FUNCTION_BLOCK INTERNAL FINAL FB_WriteRepeatedFieldInt32Tests EXTENDS FB_TestSuite
VAR_INPUT
END_VAR
VAR_OUTPUT
END_VAR
VAR
	fbFieldCodec : FB_FieldCodecInt32(nTag:= 0);
	aActual    	 : ARRAY [0..7] OF DINT;
	fbRepeatedField		: FB_RepeatedField(anyArray:= F_ToAnyType(aActual), anyFirstElem:= F_ToAnyType(aActual[0]), ipFieldCodec:= fbFieldCodec);
END_VAR

ShouldWriteRepeatedFieldTheory();

METHOD PRIVATE Reset
VAR_INPUT
END_VAR
fbRepeatedField.Initialize();
MEMSET(destAddr:= ADR(aActual), fillByte:= 16#0, n:= SIZEOF(aActual));
END_METHOD

METHOD PRIVATE ShouldWriteRepeatedField
VAR_IN_OUT CONSTANT
    aExpected   : ARRAY [*] OF BYTE;
END_VAR
VAR_INPUT
    aValues     : ARRAY [0..7] OF DINT;
    nLength     : UDINT;
    nTag        : UDINT;
    nBufferPosStart     : UDINT;
    nExpectedBufferPos  : UDINT;
    ipFieldCodec        : I_FieldCodec;
END_VAR
VAR_INST
    fbCtx   : FB_WriteContext;
END_VAR
VAR
    aActualBuffer       : ARRAY [0..63] OF BYTE;
    hr                  : HRESULT;

END_VAR
// Arrange
Reset();
fbCtx.FromBuffer(aActualBuffer);
fbCtx.refCtx.stState.nBufferPos := nBufferPosStart;
ipFieldCodec.Tag := nTag;
fbRepeatedField.InitializeFromArray(anyArray:= F_ToAnyType(aValues), anyFirstElem:= F_ToAnyType(aValues[0]), nCount:= nLength);

// Act
hr := fbRepeatedField.WriteTo(fbWriteCtx:= fbCtx, ipFieldCodec:= ipFieldCodec);

// Assert
AssertEquals_DINT(
    Expected:= S_OK,
    Actual:= hr,
    Message:= 'Expected S_OK instead of error');
    
{warning disable C0041}
AssertArrayEquals_BYTE(Expecteds:= aExpected, Actuals:= aActualBuffer, Message:= '');
 
AssertEquals_UDINT(
    Expected:= nExpectedBufferPos,
    Actual:= fbCtx.refCtx.stState.nBufferPos,
    Message:= CONCAT('Expected stState.nBufferPos to equal ', TO_STRING(nExpectedBufferPos)));
END_METHOD

METHOD PRIVATE ShouldWriteRepeatedFieldTheory : REFERENCE TO FB_Test
VAR CONSTANT
    cRawValueZeroLength     : ARRAY[0..63] OF BYTE := [16#00, 16#00];
    cRawValue1              : ARRAY[0..63] OF BYTE := [16#00, 16#0A, 16#18, 16#00, 16#D2, 16#09, 16#B9, 16#0A, 16#FF, 16#FF, 16#FF, 16#FF, 16#FF, 16#FF, 16#FF, 16#FF, 16#FF, 16#01, 16#CE, 16#C2, 16#F1, 16#05, 16#FF, 16#FF, 16#FF, 16#FF, 16#07];  
END_VAR

VAR CONSTANT
    aExpectedZeroLength     : ARRAY [0..7] OF DINT := [0, 0, 0, 0, 0, 0, 0, 0];
    aExpected1              : ARRAY [0..7] OF DINT := [0, 1234, 1337, -1, 12345678, 2147483647];
END_VAR
TEST(__POUNAME());

ShouldWriteRepeatedField(aExpected:= cRawValueZeroLength, aValues:= aExpectedZeroLength, nLength:= 0, nTag:= F_MakeTag(1, E_WireType.LengthDelimited), nBufferPosStart:= 0, nExpectedBufferPos:= 0, ipFieldCodec:= THIS^.fbFieldCodec);
ShouldWriteRepeatedField(aExpected:= cRawValue1, aValues:= aExpected1, nLength:= 6, nTag:= F_MakeTag(1, E_WireType.LengthDelimited), nBufferPosStart:= 1, nExpectedBufferPos:= 27, ipFieldCodec:= THIS^.fbFieldCodec);

TEST_FINISHED_NAMED(__POUNAME());
END_METHOD

END_FUNCTION_BLOCK

(* stored: Version 1.1.0.1
   POU FB_WriteRepeatedFieldInt32Tests: Id {bc593a6b-e6cc-4be6-a6ba-0b0aa8d4d524}, SpecialFunc None
   Method Reset: Id {1c3d5621-576c-4b6d-9236-b5891ede49f2}
   Method ShouldWriteRepeatedField: Id {320e051d-b81f-4409-b73c-7f1b4d7dc30b}
   Method ShouldWriteRepeatedFieldTheory: Id {1e79d5c0-9ca2-41ce-8d2a-0bdd3c902ca0} *)
